{attribute 'qualified_only'}
VAR_GLOBAL
	arrServoInterface		: ARRAY [1..4] OF stServoInterface;
	
	rTorqueLimit AT %Q*		: INT;
	rTorqueAct	 AT %I*		: INT;
	
	coeRead 	: FB_CoERead;
	coeWrite	: FB_CoEWrite;
	bExecute 	: BOOL;
	catchWord: INT;
END_VAR

(* stored: Version 1.1.0.1, ProductVersion 3.1.4024.12
   GVL gvlServo: Id {cc4dc48c-eb34-470f-99d5-70c06511e300} *)
